FUNCTION_BLOCK FB_Component_DualValveGuarded IMPLEMENTS I_Component
VAR_INPUT
	sName			: STRING[50];
	tTimeout		: TIME := T#0S;
END_VAR

VAR_IN_OUT
	bSensExtended	: BOOL;
	bSensRetracted	: BOOL;
	bOutputA		: BOOL;
	bOutputB		: BOOL;
END_VAR

VAR_OUTPUT
	bEnabled     	: BOOL;
	eState			: E_State;
	sStatusText 	: STRING[100];
	
	bIsExtended		: BOOL;
	bIsRetracted	: BOOL;
END_VAR

VAR
	bRetracting		: BOOL;
	bExtending		: BOOL;
	tTimeoutTimer	: TON;
	
	bLastOutputA	: BOOL;
	bLastOutputB	: BOOL;
	eLastState		: E_State;
	
	Components		: ARRAY [0..2] OF I_Component;
	
	fbPiston		: FB_Component_DualValve;
	fbReedExtended	: FB_Component_ReedSwitch;
	fbReedRetracted	: FB_Component_ReedSwitch;
END_VAR

VAR CONSTANT
	DISABLED		: E_State := E_State.DISABLED;
	READY			: E_State := E_State.READY;
	BUSY			: E_State := E_State.BUSY;
	DONE			: E_State := E_State.DONE;
	HALTED			: E_State := E_State.HALTED;
	TIMEOUT			: E_State := E_State.TIMEOUT;
END_VAR

tTimeoutTimer(PT := tTimeout);

fbPiston(sName := '', tTimeout 	:= T#0S, bOutputA := bOutputA, bOutputB := bOutputB);
fbReedExtended(sName := '', bRawSignal 	:= bSensExtended, tTimeout := T#0S);
fbReedRetracted(sName := '', bRawSignal 	:= bSensRetracted, tTimeout := T#0S);

Components[0] := fbPiston;
Components[1] := fbReedExtended;
Components[2] := fbReedRetracted;

bIsExtended		:= fbReedExtended.bSensorActive;
bIsRetracted	:= fbReedRetracted.bSensorActive;

CASE eState OF
	DISABLED: 	sStatusText := 'piston disabled';
	READY: 		sStatusText :=  CONCAT(CONCAT(SEL(bIsExtended = TRUE, '', 'piston extended and '),SEL(bIsRetracted = TRUE, '', 'piston retracted and ')), 'ready to operate');
	
	BUSY: 		IF bExtending THEN
					sStatusText := 'piston extending';
					IF fbReedExtended.bSensorActive THEN
						fbPiston.M_Hold();
						eState := TIMEOUT;
					ELSE
						fbPiston.M_Extend();
					END_IF
				END_IF
				IF bRetracting THEN
					sStatusText := 'piston retracting';
					IF fbReedRetracted.bSensorActive THEN
						fbPiston.M_Hold();
						eState := TIMEOUT;
					ELSE
						fbPiston.M_Retract();
					END_IF
				END_IF
			
	TIMEOUT:	sStatusText := 'piston in timeout';
				bExtending  := FALSE;
				bRetracting := FALSE;
				tTimeoutTimer(IN := TRUE);
				
				IF tTimeoutTimer.Q THEN
					eState := E_State.DONE;
				END_IF
				
	DONE:		sStatusText := 'piston done';
				tTimeoutTimer(IN := FALSE);
				M_Resume();
				
	HALTED:		sStatusText := 'piston halted';
END_CASE

{warning 'add method implementation '}
METHOD M_Disable : BOOL
VAR
	idx	: INT := 0;
END_VAR
IF eState = DONE OR eState = READY THEN
	bEnabled	:= FALSE;
	eState		:= DISABLED;
	
	FOR idx := 0 TO 2 DO
    	Components[idx].M_Disable();
	END_FOR;
END_IF
END_METHOD

{warning 'add method implementation '}
METHOD M_Enable : BOOL

VAR
	idx: INT;
END_VAR
IF eState = DISABLED THEN
	bEnabled	:= TRUE;
	eState 		:= READY;
	
	FOR idx := 0 TO 2 DO
    	Components[idx].M_Enable();
	END_FOR;
END_IF
END_METHOD

METHOD M_Extend : BOOL
VAR_INPUT
END_VAR
IF eState = READY AND NOT fbReedExtended.bSensorActive THEN
	bExtending 	:= TRUE;
	eState 		:= BUSY;
END_IF
END_METHOD

{warning 'add method implementation '}
METHOD M_Halt : BOOL
bLastOutputA 	:= bOutputA;
bLastOutputB 	:= bOutputB;
bOutputA		:= FALSE;
bOutputB		:= FALSE;
eLastState 		:= eState;
eState 			:= HALTED;
END_METHOD

{warning 'add method implementation '}
METHOD M_Reset : BOOL
END_METHOD

{warning 'add method implementation '}
METHOD M_Resume : BOOL

VAR
	idx: INT;
END_VAR
CASE eState OF
	DISABLED:	eState 		:= eLastState;
				bOutputA 	:= bLastOutputA;
				bOutputB 	:= bLastOutputB;
				FOR idx := 0 TO 2 DO
					Components[idx].M_Resume();
				END_FOR;
				
	DONE:		eState := READY;
END_CASE
END_METHOD

METHOD M_Retract : BOOL
VAR_INPUT
END_VAR
IF eState = READY AND NOT fbReedRetracted.bSensorActive  THEN
	bRetracting	:= TRUE;
	eState 		:= BUSY;
END_IF
END_METHOD

{warning 'add method implementation '}
METHOD M_Stop : BOOL

VAR
	idx: INT := 0;
END_VAR
IF eState = READY OR eState = DONE THEN
	eState := DONE;
	
	FOR idx := 0 TO 2 DO
    	Components[idx].M_Stop();
	END_FOR;
END_IF
END_METHOD

END_FUNCTION_BLOCK

(* stored: Version 1.1.0.1, ProductVersion 3.1.4024.15
   POU FB_Component_DualValveGuarded: Id {c556a97c-7b93-4813-959c-89767b9fff4c}, SpecialFunc None
   Method M_Disable: Id {87f5b470-e1c8-47c8-8841-531e8d9726b2}
   Method M_Enable: Id {d6b033a0-41c9-498d-b55b-6168c29d2e9a}
   Method M_Extend: Id {349c74e4-2aba-4161-a448-723bfc73a6ee}
   Method M_Halt: Id {738271be-bd18-41db-b217-73aa834901fc}
   Method M_Reset: Id {1329416a-ff99-4d41-b874-81ccef35708a}
   Method M_Resume: Id {b6b32c60-781e-4ba1-a85a-eed5180e722d}
   Method M_Retract: Id {5299460a-3373-4e48-9b38-fc81c8faba27}
   Method M_Stop: Id {30525d9f-a584-4e50-bd95-dc81937f8e2d} *)
